// TIA Portal V15.1 export
// export: Created 2024-05-17T05:38:43.6338741Z, ExportSetting WithDefaults, DisplayName Totally Integrated Automation Portal, DisplayVersion V15.1 Update 5, DisplayName TIA Portal Openness, DisplayVersion V15.1 Update 5, DisplayName SINAMICS Startdrive Advanced, DisplayVersion V15.1, DisplayName G130, G150, S120, S150, SINAMICS MV, S210, DisplayVersion V15.1, DisplayName G110M, G120, G120C, G120D, G120P, DisplayVersion V15.1, DisplayName STEP 7 Professional, DisplayVersion V15.1 Update 5, DisplayName STEP 7 Safety, DisplayVersion V15.1, DisplayName WinCC Professional, DisplayVersion V15.1 Update 5, DisplayName SIMATIC Visualization Architect, DisplayVersion V15.1
FUNCTION "LGBValveStatusSub" : Void   // FC6604, FBD
TITLE = LGBValveStatusSub
{ S7_Optimized_Access := 'TRUE' }
VERSION : 0.1
// stored: AutoNumber false, IsIECCheckEnabled false, SetENOAutomatically False, UDAEnableTagReadback false
   VAR_INPUT
      PipeData : "TCPipe";
   END_VAR
   VAR_OUTPUT
      ValveStatus : "TCValve";
   END_VAR
BEGIN

REGION Network 1: Valve not used IBC 1
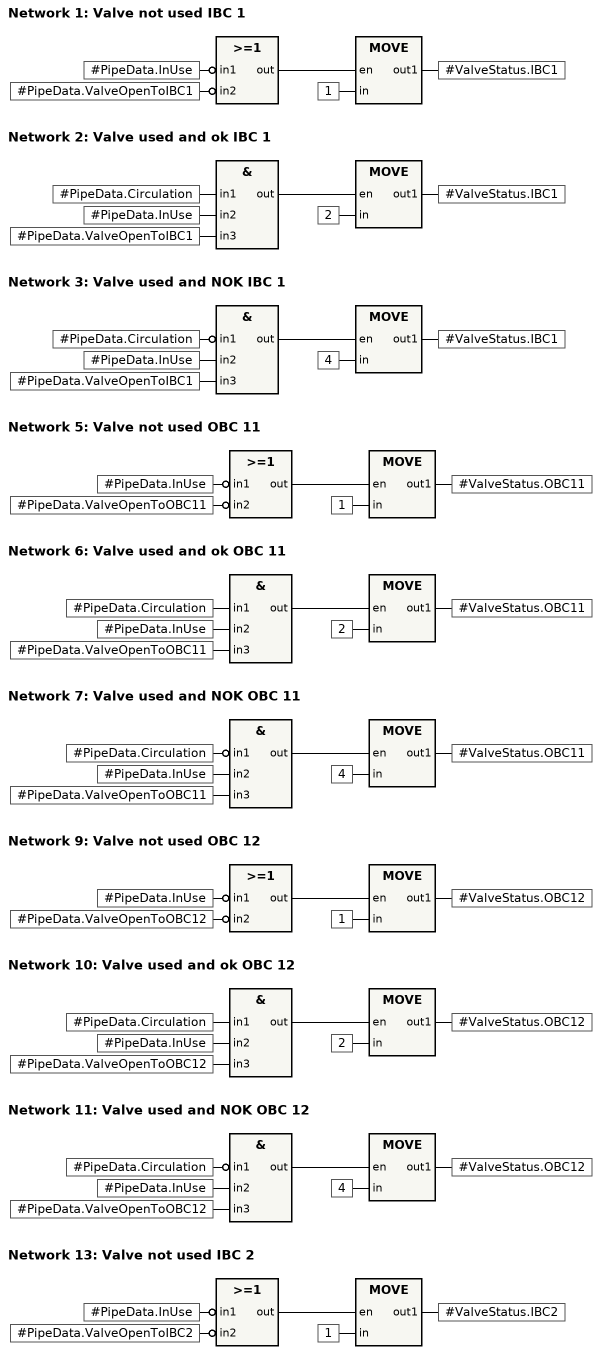
   IF NOT #PipeData.InUse OR NOT #PipeData.ValveOpenToIBC1 THEN #ValveStatus.IBC1 := 1; END_IF;
END_REGION

REGION Network 2: Valve used and ok IBC 1
   IF #PipeData.Circulation AND #PipeData.InUse AND #PipeData.ValveOpenToIBC1 THEN
       #ValveStatus.IBC1 := 2;
   END_IF;
END_REGION

REGION Network 3: Valve used and NOK IBC 1
   IF NOT #PipeData.Circulation AND #PipeData.InUse AND #PipeData.ValveOpenToIBC1 THEN
       #ValveStatus.IBC1 := 4;
   END_IF;
END_REGION

REGION Network 5: Valve not used OBC 11
   IF NOT #PipeData.InUse OR NOT #PipeData.ValveOpenToOBC11 THEN #ValveStatus.OBC11 := 1; END_IF;
END_REGION

REGION Network 6: Valve used and ok OBC 11
   IF #PipeData.Circulation AND #PipeData.InUse AND #PipeData.ValveOpenToOBC11 THEN
       #ValveStatus.OBC11 := 2;
   END_IF;
END_REGION

REGION Network 7: Valve used and NOK OBC 11
   IF NOT #PipeData.Circulation AND #PipeData.InUse AND #PipeData.ValveOpenToOBC11 THEN
       #ValveStatus.OBC11 := 4;
   END_IF;
END_REGION

REGION Network 9: Valve not used OBC 12
   IF NOT #PipeData.InUse OR NOT #PipeData.ValveOpenToOBC12 THEN #ValveStatus.OBC12 := 1; END_IF;
END_REGION

REGION Network 10: Valve used and ok OBC 12
   IF #PipeData.Circulation AND #PipeData.InUse AND #PipeData.ValveOpenToOBC12 THEN
       #ValveStatus.OBC12 := 2;
   END_IF;
END_REGION

REGION Network 11: Valve used and NOK OBC 12
   IF NOT #PipeData.Circulation AND #PipeData.InUse AND #PipeData.ValveOpenToOBC12 THEN
       #ValveStatus.OBC12 := 4;
   END_IF;
END_REGION

REGION Network 13: Valve not used IBC 2
   IF NOT #PipeData.InUse OR NOT #PipeData.ValveOpenToIBC2 THEN #ValveStatus.IBC2 := 1; END_IF;
END_REGION

REGION Network 14: Valve used and ok IBC 2
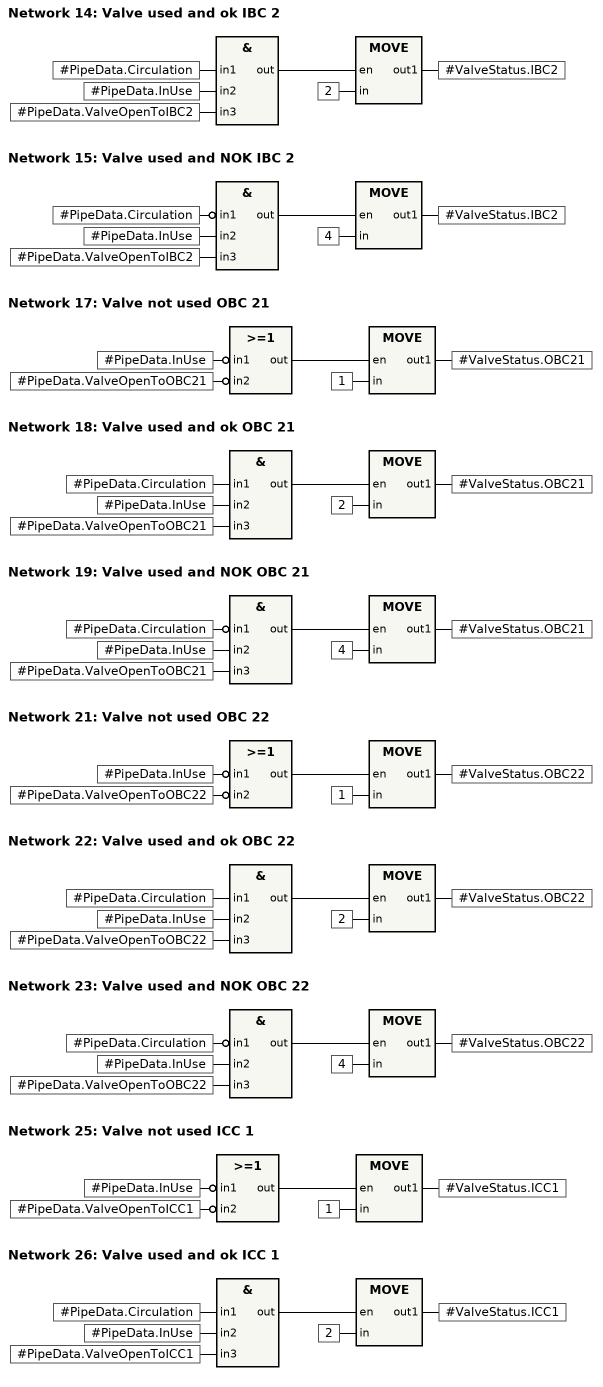
   IF #PipeData.Circulation AND #PipeData.InUse AND #PipeData.ValveOpenToIBC2 THEN
       #ValveStatus.IBC2 := 2;
   END_IF;
END_REGION

REGION Network 15: Valve used and NOK IBC 2
   IF NOT #PipeData.Circulation AND #PipeData.InUse AND #PipeData.ValveOpenToIBC2 THEN
       #ValveStatus.IBC2 := 4;
   END_IF;
END_REGION

REGION Network 17: Valve not used OBC 21
   IF NOT #PipeData.InUse OR NOT #PipeData.ValveOpenToOBC21 THEN #ValveStatus.OBC21 := 1; END_IF;
END_REGION

REGION Network 18: Valve used and ok OBC 21
   IF #PipeData.Circulation AND #PipeData.InUse AND #PipeData.ValveOpenToOBC21 THEN
       #ValveStatus.OBC21 := 2;
   END_IF;
END_REGION

REGION Network 19: Valve used and NOK OBC 21
   IF NOT #PipeData.Circulation AND #PipeData.InUse AND #PipeData.ValveOpenToOBC21 THEN
       #ValveStatus.OBC21 := 4;
   END_IF;
END_REGION

REGION Network 21: Valve not used OBC 22
   IF NOT #PipeData.InUse OR NOT #PipeData.ValveOpenToOBC22 THEN #ValveStatus.OBC22 := 1; END_IF;
END_REGION

REGION Network 22: Valve used and ok OBC 22
   IF #PipeData.Circulation AND #PipeData.InUse AND #PipeData.ValveOpenToOBC22 THEN
       #ValveStatus.OBC22 := 2;
   END_IF;
END_REGION

REGION Network 23: Valve used and NOK OBC 22
   IF NOT #PipeData.Circulation AND #PipeData.InUse AND #PipeData.ValveOpenToOBC22 THEN
       #ValveStatus.OBC22 := 4;
   END_IF;
END_REGION

REGION Network 25: Valve not used ICC 1
   IF NOT #PipeData.InUse OR NOT #PipeData.ValveOpenToICC1 THEN #ValveStatus.ICC1 := 1; END_IF;
END_REGION

REGION Network 26: Valve used and ok ICC 1
   IF #PipeData.Circulation AND #PipeData.InUse AND #PipeData.ValveOpenToICC1 THEN
       #ValveStatus.ICC1 := 2;
   END_IF;
END_REGION

REGION Network 27: Valve used and NOK ICC 1
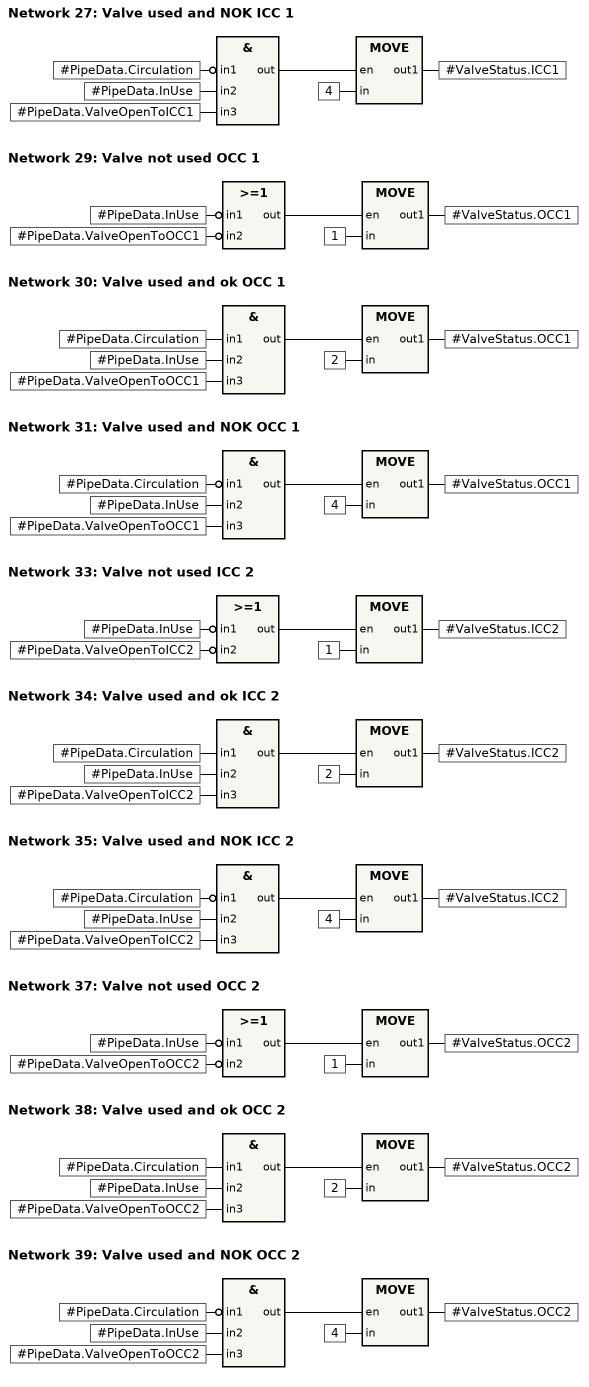
   IF NOT #PipeData.Circulation AND #PipeData.InUse AND #PipeData.ValveOpenToICC1 THEN
       #ValveStatus.ICC1 := 4;
   END_IF;
END_REGION

REGION Network 29: Valve not used OCC 1
   IF NOT #PipeData.InUse OR NOT #PipeData.ValveOpenToOCC1 THEN #ValveStatus.OCC1 := 1; END_IF;
END_REGION

REGION Network 30: Valve used and ok OCC 1
   IF #PipeData.Circulation AND #PipeData.InUse AND #PipeData.ValveOpenToOCC1 THEN
       #ValveStatus.OCC1 := 2;
   END_IF;
END_REGION

REGION Network 31: Valve used and NOK OCC 1
   IF NOT #PipeData.Circulation AND #PipeData.InUse AND #PipeData.ValveOpenToOCC1 THEN
       #ValveStatus.OCC1 := 4;
   END_IF;
END_REGION

REGION Network 33: Valve not used ICC 2
   IF NOT #PipeData.InUse OR NOT #PipeData.ValveOpenToICC2 THEN #ValveStatus.ICC2 := 1; END_IF;
END_REGION

REGION Network 34: Valve used and ok ICC 2
   IF #PipeData.Circulation AND #PipeData.InUse AND #PipeData.ValveOpenToICC2 THEN
       #ValveStatus.ICC2 := 2;
   END_IF;
END_REGION

REGION Network 35: Valve used and NOK ICC 2
   IF NOT #PipeData.Circulation AND #PipeData.InUse AND #PipeData.ValveOpenToICC2 THEN
       #ValveStatus.ICC2 := 4;
   END_IF;
END_REGION

REGION Network 37: Valve not used OCC 2
   IF NOT #PipeData.InUse OR NOT #PipeData.ValveOpenToOCC2 THEN #ValveStatus.OCC2 := 1; END_IF;
END_REGION

REGION Network 38: Valve used and ok OCC 2
   IF #PipeData.Circulation AND #PipeData.InUse AND #PipeData.ValveOpenToOCC2 THEN
       #ValveStatus.OCC2 := 2;
   END_IF;
END_REGION

REGION Network 39: Valve used and NOK OCC 2
   IF NOT #PipeData.Circulation AND #PipeData.InUse AND #PipeData.ValveOpenToOCC2 THEN
       #ValveStatus.OCC2 := 4;
   END_IF;
END_REGION
END_FUNCTION
